METHOD PUBLIC GetSerializer : I_Serializer
VAR_INPUT
END_VAR
GetSerializer := serializer.Clone();
END_METHOD

METHOD PUBLIC RejectWithError
VAR_INPUT
	ErrorCode : T_MAXSTRING;
	Message : T_MAXSTRING;
END_VAR
serverResponse.Error(ErrorCode, Message);
END_METHOD

METHOD PUBLIC TryMakeAsynchronous : BOOL
VAR_INPUT
	Destination : REFERENCE TO I_AsynchronousRpcResponse;
END_VAR
VAR
	asynchronousRpcResponseFactory : AsynchronousRpcResponseFactory(serverResponse, serializer, asyncResponseManager);
END_VAR
TryMakeAsynchronous := asynchronousRpcResponseFactory.TryCreate(Destination);
END_METHOD

END_FUNCTION_BLOCK

// _Internal/RPC/Response/Factory/AsynchronousRpcResponseFactory
{attribute 'linkalways'} 
{attribute 'no_explicit_call' := 'This FB is a CLASS and must be accessed using methods or properties'}
{attribute 'enable_dynamic_creation'}
FUNCTION_BLOCK AsynchronousRpcResponseFactory IMPLEMENTS I_AsynchronousRpcResponseFactory
VAR
	serverResponse : I_ServerResponse;
	serializer : I_Serializer;
	asyncResponseManager : I_AsyncResponseManager;
END_VAR

METHOD FB_init : BOOL
VAR_INPUT
	bInitRetains : BOOL; // if TRUE, the retain variables are initialized (warm start / cold start)
	bInCopyCode : BOOL;  // if TRUE, the instance afterwards gets moved into the copy code (online change)
	ServerResponse : I_ServerResponse;
	Serializer : I_Serializer;
	AsyncResponseManager : I_AsyncResponseManager;
END_VAR
THIS^.serverResponse := ServerResponse;
THIS^.serializer := Serializer;
THIS^.asyncResponseManager := AsyncResponseManager;
END_METHOD

METHOD PUBLIC TryCreate : BOOL
VAR_INPUT
	Destination : REFERENCE TO I_AsynchronousRpcResponse;
END_VAR
VAR
	asyncResponseSessionData : I_AsyncResponseSessionData;
	pAsynchronousRpcResponse : POINTER TO AsynchronousRpcResponse;
END_VAR
IF NOT asyncResponseManager.TryConvertResponseToAsyncResponseSessionData(serverResponse, 0, asyncResponseSessionData) THEN
	RETURN;
END_IF

pAsynchronousRpcResponse := __NEW(AsynchronousRpcResponse(AsyncResponse := asyncResponseSessionData, Serializer := THIS^.serializer));
Destination := pAsynchronousRpcResponse^;
TryCreate := TRUE;
END_METHOD

END_FUNCTION_BLOCK

// _Internal/RPC/Response/Factory/I_AsynchronousRpcResponseFactory
INTERFACE I_AsynchronousRpcResponseFactory

METHOD PUBLIC TryCreate : BOOL
VAR_INPUT
	Destination : REFERENCE TO I_AsynchronousRpcResponse;
END_VAR
END_METHOD

END_INTERFACE

// _Internal/RPC/Middleware/RpcMiddleware
{attribute 'linkalways'} 
{attribute 'no_explicit_call' := 'This FB is a CLASS and must be accessed using methods or properties'}
{attribute 'enable_dynamic_creation'}
FUNCTION_BLOCK RpcMiddleware EXTENDS MiddlewareBase
VAR
	rpcManager : I_RpcManager;
END_VAR

METHOD FB_init : BOOL
VAR_INPUT
	bInitRetains : BOOL; // if TRUE, the retain variables are initialized (warm start / cold start)
	bInCopyCode : BOOL;  // if TRUE, the instance afterwards gets moved into the copy code (online change)
	RpcManager : I_RpcManager;
END_VAR
THIS^.rpcManager := RpcManager;
END_METHOD

METHOD PUBLIC Handle
VAR_INPUT
	Request : I_Request;
	Response : I_ServerResponse;
END_VAR
IF rpcManager.TryHandleIncomingRequest(Request, Response) THEN
	RETURN;
END_IF

Next(Request, Response);
END_METHOD

END_FUNCTION_BLOCK

// _Internal/RPC/RegisteredRpcApis/RegisteredRpcApis
{attribute 'linkalways'} 
{attribute 'no_explicit_call' := 'This FB is a CLASS and must be accessed using methods or properties'}
{attribute 'enable_dynamic_creation'}
FUNCTION_BLOCK RegisteredRpcApis
VAR
	registeredRpcApis : Queue;
	_hasRegisteredRpcApis : BOOL;
	enumerator : I_ForwardEnumerator;
END_VAR

METHOD FB_exit : BOOL
VAR_INPUT
	bInCopyCode : BOOL; // if TRUE, the exit method is called for exiting an instance that is copied afterwards (online change).
END_VAR
IF bInCopyCode THEN
	RETURN;
END_IF

IF enumerator <> 0 THEN
	enumerator.Dispose();
END_IF
END_METHOD

METHOD PRIVATE CreateEnumerator
VAR_INPUT
END_VAR
IF enumerator <> 0 THEN
	enumerator.Dispose();
END_IF

enumerator := registeredRpcApis.GetEnumerator();
END_METHOD

METHOD PUBLIC CyclicCall
VAR
	rpcApi : I_RpcApi;
END_VAR
IF NOT HasRegisteredRpcApis THEN
	RETURN;
END_IF

enumerator.Reset();

WHILE enumerator.MoveNext() DO
	IF enumerator.TryGet(rpcApi) THEN
		rpcApi.CyclicCall();
	END_IF;
END_WHILE
END_METHOD

PROPERTY PUBLIC HasRegisteredRpcApis : BOOL
GET
HasRegisteredRpcApis := enumerator <> 0;
END_GET
END_PROPERTY

METHOD PUBLIC RegisterRpcApi
VAR_INPUT
	RpcApi : I_RpcApi;
END_VAR
registeredRpcApis.Enqueue(RpcApi);
CreateEnumerator();
END_METHOD

END_FUNCTION_BLOCK

// RpcApi/I_RpcApi
INTERFACE I_RpcApi

METHOD CyclicCall
VAR_INPUT
END_VAR
END_METHOD

METHOD RegisterAsynchronousRpcHandlersWith
VAR_INPUT
	Host : I_HostAsynchronousRpcHandlers;
END_VAR
END_METHOD

METHOD RegisterSynchronousRpcHandlersWith
VAR_INPUT
	Host : I_HostSynchronousRpcHandlers;
END_VAR
END_METHOD

END_INTERFACE

// _Internal/Sessions/Manager/I_SessionManager
INTERFACE I_SessionManager

METHOD PUBLIC CreateSession : T_MAXSTRING
END_METHOD

METHOD PUBLIC DisposeAllSessions
VAR_INPUT
END_VAR
END_METHOD

METHOD PUBLIC IsValidSession : BOOL
VAR_INPUT
	Id : T_MAXSTRING;
END_VAR
END_METHOD

METHOD PUBLIC RefreshSession
VAR_INPUT
	Id : T_MAXSTRING;
END_VAR
END_METHOD

END_INTERFACE

// _Internal/Sessions/Manager/SessionManager
{attribute 'linkalways'} 
{attribute 'no_explicit_call' := 'This FB is a CLASS and must be accessed using methods or properties'}
{attribute 'enable_dynamic_creation'}
FUNCTION_BLOCK SessionManager implements I_SessionManager, I_SessionStorage
VAR
	activeSessions : Dictionary;
	sessionIdGenerator : I_SessionIdGenerator;
	currentStorageId : UDINT;
	sessionMaxLife : TIME;
END_VAR

METHOD FB_init : BOOL
VAR_INPUT
	bInitRetains : BOOL; // if TRUE, the retain variables are initialized (warm start / cold start)
	bInCopyCode : BOOL;  // if TRUE, the instance afterwards gets moved into the copy code (online change)
	SessionIdGenerator : I_SessionIdGenerator;
	SessionMaxLife : TIME;
END_VAR
THIS^.sessionIdGenerator := SessionIdGenerator;
THIS^.sessionMaxLife := SessionMaxLife;
END_METHOD

METHOD FB_exit : BOOL
VAR_INPUT
	bInCopyCode : BOOL; // if TRUE, the exit method is called for exiting an instance that is copied afterwards (online change).
END_VAR
IF bInCopyCode THEN
	RETURN;
END_IF

DisposeAllSessions();
END_METHOD

METHOD PUBLIC CheckForExpiredSessions
VAR_INPUT
END_VAR
VAR
	enumerator : I_ForwardEnumerator;
	session : I_Session;
	expiredSessions : Stack;
END_VAR
enumerator := activeSessions.GetEnumerator();

WHILE enumerator.MoveNext() DO
	IF enumerator.TryGet(session) THEN
		IF session.LastAccessedTimestamp.IsDurationElapsed(sessionMaxLife) THEN
			expiredSessions.Push(session);
		END_IF
	END_IF
END_WHILE

enumerator.Dispose();

WHILE expiredSessions.TryPop(session) DO
	DisposeSession(session.Id);
END_WHILE
END_METHOD

METHOD PRIVATE CreateNewSession : I_Session
VAR
	id : T_MAXSTRING;
	pSession : POINTER TO Session;
END_VAR
id := sessionIdGenerator.Generate();
pSession := __NEW(Session(SessionId := id));
CreateNewSession := pSession^;
END_METHOD

METHOD PUBLIC CreateSession : T_MAXSTRING;
VAR
	session : I_Session;
END_VAR
session := CreateNewSession();
activeSessions.AddOrUpdate(session.Id, session);
CreateSession := session.Id;
END_METHOD

METHOD PUBLIC CyclicCall
VAR_INPUT
END_VAR
CheckForExpiredSessions();
END_METHOD

METHOD PUBLIC DisposeAllSessions
VAR_INPUT
END_VAR
VAR
	enumerator : I_ForwardEnumerator;
	session : I_Session;
END_VAR
enumerator := activeSessions.GetEnumerator();

WHILE enumerator.MoveNext() DO
	if enumerator.TryGet(session) then
		session.Dispose();
	END_IF
END_WHILE

enumerator.Dispose();
activeSessions.Clear();
END_METHOD

METHOD PUBLIC DisposeSession
VAR_INPUT
	Id : T_MAXSTRING;
END_VAR
VAR
	session : I_Session;
END_VAR
IF NOT activeSessions.TryGetValue(Id, session) THEN
	RETURN;
END_IF

session.Dispose();
activeSessions.Remove(Id);
END_METHOD

METHOD PUBLIC DisposeSessionDataById
VAR_INPUT
	SessionId : T_MAXSTRING;
	StorageId : T_MAXSTRING;
END_VAR
VAR
	session : I_Session;
	sessionData : I_SessionData;
END_VAR
IF StorageId = '' THEN 
	RETURN;
END_IF

IF NOT activeSessions.TryGetValue(SessionId, session) THEN
	RETURN;
END_IF

IF NOT session.TryGetDataFromStorage(StorageId, sessionData) THEN
	RETURN;
END_IF

session.DisposeDataFromStorage(StorageId);
END_METHOD

METHOD PUBLIC IsValidSession : BOOL
VAR_INPUT
	Id : T_MAXSTRING;
END_VAR
IsValidSession := activeSessions.ContainsKey(Id);
END_METHOD

METHOD PUBLIC RefreshSession
VAR_INPUT
	Id : T_MAXSTRING;
END_VAR
VAR
	session : I_Session;
END_VAR
IF NOT activeSessions.TryGetValue(Id, session) THEN
	RETURN;
END_IF

session.Refresh();
END_METHOD

PROPERTY PUBLIC SessionCount : DINT
GET
SessionCount := activeSessions.Count;
END_GET
END_PROPERTY

METHOD PUBLIC TryRetreiveSessionDataById : BOOL
VAR_INPUT
	SessionId : T_MAXSTRING;
	StorageId : T_MAXSTRING;
	Destination : REFERENCE TO I_SessionData;
END_VAR
VAR
	session : I_Session;
END_VAR
IF NOT activeSessions.TryGetValue(SessionId, session) THEN
	RETURN;
END_IF

TryRetreiveSessionDataById := session.TryGetDataFromStorage(StorageId, Destination);
END_METHOD

METHOD PUBLIC TryStoreSessionDataById : BOOL
VAR_INPUT
	SessionId : T_MAXSTRING;
	StorageId : T_MAXSTRING;
	Source : I_SessionData;
END_VAR
VAR
	session : I_Session;
END_VAR
IF StorageId = '' THEN 
	RETURN;
END_IF

IF NOT activeSessions.TryGetValue(SessionId, session) THEN
	RETURN;
END_IF

session.AddOrUpdateStorage(StorageId, Source);
TryStoreSessionDataById := TRUE;
END_METHOD

END_FUNCTION_BLOCK

// _Internal/Sessions/SessionId/I_SessionIdGenerator
INTERFACE I_SessionIdGenerator

METHOD PUBLIC Generate : T_MAXSTRING
VAR_INPUT
END_VAR
END_METHOD

END_INTERFACE

// _Internal/Sessions/Middleware/SessionsMiddleware
{attribute 'linkalways'} 
{attribute 'no_explicit_call' := 'This FB is a CLASS and must be accessed using methods or properties'}
{attribute 'enable_dynamic_creation'}
FUNCTION_BLOCK SessionsMiddleware EXTENDS MiddlewareBase
VAR
	sessionManager: I_SessionManager;
	headerAccessor : I_SessionHeaderAccessor;
END_VAR

METHOD FB_init : BOOL
VAR_INPUT
	bInitRetains : BOOL; // if TRUE, the retain variables are initialized (warm start / cold start)
	bInCopyCode : BOOL;  // if TRUE, the instance afterwards gets moved into the copy code (online change)
	SessionManager : I_SessionManager;
	HeaderAccessor : I_SessionHeaderAccessor;
END_VAR
THIS^.sessionManager := SessionManager;
THIS^.headerAccessor := HeaderAccessor;
END_METHOD

METHOD PUBLIC Handle
VAR_INPUT
	Request : I_Request;
	Response : I_ServerResponse;
END_VAR
VAR
	sessionId : T_MAXSTRING;
END_VAR
IF (NOT headerAccessor.TryGetSessionIdFromRequest(Request, sessionId)) OR_ELSE (NOT sessionManager.IsValidSession(sessionId)) THEN
	sessionId := sessionManager.CreateSession();
	headerAccessor.UpdateRequestWithSessionId(Request,sessionId);
END_IF

sessionManager.RefreshSession(sessionId);

headerAccessor.UpdateResponseWithSessionId(Response, sessionId);
Next(Request, Response);
END_METHOD

END_FUNCTION_BLOCK

// _Internal/Sessions/SessionId/SequentialSessionIdGenerator
{attribute 'linkalways'} 
{attribute 'no_explicit_call' := 'This FB is a CLASS and must be accessed using methods or properties'}
{attribute 'enable_dynamic_creation'}
FUNCTION_BLOCK SequentialSessionIdGenerator Implements I_SessionIdGenerator
VAR
	currentCount : UDINT;
END_VAR

METHOD PUBLIC Generate : T_MAXSTRING
VAR_INPUT
END_VAR
currentCount := currentCount + 1;
Generate := UDINT_TO_STRING(currentCount);
END_METHOD

END_FUNCTION_BLOCK

// RpcHandler/Examples/AsyncConcatStringRpcHandler
{attribute 'linkalways'} 
FUNCTION_BLOCK AsyncConcatStringRpcHandler IMPLEMENTS I_AsynchronousRpcHandler
VAR
END_VAR

METHOD Handle
VAR_INPUT
	Parameters : I_Deserializer;
	Response : I_AsynchronousRpcResponse;
END_VAR
VAR
	str1 : T_MAXSTRING;
	str2 : T_MAXSTRING;
	result : T_MAXSTRING;
	feedback : DeserializerFeedback;
END_VAR
IF NOT Parameters.TryGetKeyString('STR1',str1,feedback) THEN
	Response.RejectWithError('MISSING_PARAMETER',feedback.FirstError.Message);
	RETURN;
END_IF

IF NOT Parameters.TryGetKeyString('STR2',str2,feedback) THEN
	Response.RejectWithError('MISSING_PARAMETER',feedback.FirstError.Message);
	RETURN;
END_IF

result := CONCAT(str1, str2);
Response.CompleteWithString(result);
END_METHOD

END_FUNCTION_BLOCK

// RpcHandler/Examples/ConcatStringRpcHandler
{attribute 'linkalways'} 
FUNCTION_BLOCK ConcatStringRpcHandler IMPLEMENTS I_SynchronousRpcHandler
VAR
END_VAR

METHOD Handle
VAR_INPUT
	Parameters : I_Deserializer;
	Response : I_SynchronousRpcResponse;
END_VAR
VAR
	str1 : T_MAXSTRING;
	str2 : T_MAXSTRING;
	result : T_MAXSTRING;
	feedback : DeserializerFeedback;
END_VAR
IF NOT Parameters.TryGetKeyString('STR1',str1,feedback) THEN
	Response.RejectWithError('MISSING_PARAMETER',feedback.FirstError.Message);
	RETURN;
END_IF

IF NOT Parameters.TryGetKeyString('STR2',str2,feedback) THEN
	Response.RejectWithError('MISSING_PARAMETER',feedback.FirstError.Message);
	RETURN;
END_IF

result := CONCAT(str1, str2);
Response.CompleteWithString(result);
END_METHOD

END_FUNCTION_BLOCK

// RpcServer/I_RpcServer
INTERFACE I_RpcServer

METHOD PUBLIC GetConfiguredHeaderSize : UDINT
VAR_INPUT
END_VAR
END_METHOD

METHOD PUBLIC GetConfiguredPayloadSize : UDINT
VAR_INPUT
END_VAR
END_METHOD

{attribute 'TcRpcEnable'}
METHOD PUBLIC HandleRequest : ResponseData;
VAR_INPUT
	SerializedHeader : STRING(ServerConfiguration.HEADER_STRING_SIZE);
	SerializedPayload : STRING(ServerConfiguration.PAYLOAD_STRING_SIZE);
END_VAR
END_METHOD

METHOD PUBLIC RegisterApi
VAR_INPUT
	RpcApi : I_RpcApi;
END_VAR
END_METHOD

METHOD PUBLIC RegisterAsynchronousRpcHandler
VAR_INPUT
	MethodName : T_MAXSTRING;
	Handler : I_AsynchronousRpcHandler;
END_VAR
END_METHOD

METHOD PUBLIC RegisterSynchronousRpcHandler
VAR_INPUT
	MethodName : T_MAXSTRING;
	Handler : I_SynchronousRpcHandler;
END_VAR
END_METHOD

END_INTERFACE

// RpcServer/RpcServer
{attribute 'linkalways'} 
{attribute 'no_explicit_call' := 'This FB is a CLASS and must be accessed using methods or properties'}
{attribute 'enable_dynamic_creation'}
{attribute 'TcRpcEnable'}
FUNCTION_BLOCK RpcServer IMPLEMENTS I_RpcServer
VAR
	// default header accessor.
	headerAccessor : HeaderAccessor;
	
	// Payload size may be changed using the constants
	payloadStringSizeIncludingNull : UDINT := ServerConfiguration.PAYLOAD_STRING_SIZE + 1;
	
	// the middleware stack allows us to construct our server in any way needed.
	// by default we will support sessions, async polling and chunked requests/
	middlewareStack : MiddlewareStack;
	
	// responseId generation required for pending or chunked data
	sequentialResponseIdGenerator : SequentialResponseIdGenerator;
	
	// ability to support sessions...
	sessionIdGenerator : SequentialSessionIdGenerator;
	sessionManager : SessionManager(sessionIdGenerator, INACTIVE_SESSION_MAX_AGE);
	sessionsMiddleware : SessionsMiddleware(sessionManager, headerAccessor);
	
	// ability to suppoort chunked requests
	chunkedRequestsManager : ChunkedRequestsManager(payloadStringSizeIncludingNull, sessionManager, headerAccessor);
	chunkedRequestsMiddleware : ChunkedRequestsMiddleware(chunkedRequestsManager);
	
	// ability to support chunked responses
	chunkedResponseManager : ChunkedResponseManager(payloadStringSizeIncludingNull, sessionManager, sequentialResponseIdGenerator, headerAccessor);
	chunkedResponsesMiddleware : ChunkedResponsesMiddleware(chunkedResponseManager);
	
	// ability to support pending responses
	asyncResponseManager : AsyncResponseManager(sessionManager, sequentialResponseIdGenerator, headerAccessor);
	asyncResponseMiddleware : AsyncResponseMiddleware(asyncResponseManager);
	
	// ability to support rpc
	synchronousRpcHandlers : SynchronousRpcHandlers;
	asynchronousRpcHandlers : AsynchronousRpcHandlers;
	asyncRpcCallQueue : AsyncRpcCallQueue;
	rpcManager : RpcManager(synchronousRpcHandlers, asynchronousRpcHandlers, asyncResponseManager, headerAccessor, asyncRpcCallQueue);
	rpcMiddleware : RpcMiddleware(rpcManager);
	
	// registered apis (used for cyclic calling)
	registeredRpcApis : RegisteredRpcApis;
	
END_VAR
VAR CONSTANT
	INACTIVE_SESSION_MAX_AGE : TIME := T#10S;
END_VAR

METHOD FB_init : BOOL
VAR_INPUT
	bInitRetains : BOOL; // if TRUE, the retain variables are initialized (warm start / cold start)
	bInCopyCode : BOOL;  // if TRUE, the instance afterwards gets moved into the copy code (online change)
END_VAR
// must be above any middleware which requires storing of session data. 
// best practice is to put at the top
MiddlewareStack.Use(sessionsMiddleware);

// must be above any middleware which could send a response larger than the max payload.
// once this is in place then middleware can send as large as they like (up to router memory max)
MiddlewareStack.Use(chunkedResponsesMiddleware);

// must be above any middleware which needs to support async responses
MiddlewareStack.Use(AsyncResponseMiddleware);

// chunked request must be after chunked response to prevent incorrectly starting a new request
// if the client askes for a response without removing the last request header.
MiddlewareStack.Use(chunkedRequestsMiddleware); 

// rpc middlware.  All other middleware can go under here.
MiddlewareStack.Use(rpcMiddleware);
END_METHOD

METHOD PUBLIC CyclicCall
VAR_INPUT
END_VAR
sessionManager.CyclicCall();
asyncRpcCallQueue.CyclicCall();
registeredRpcApis.CyclicCall();
END_METHOD

{attribute 'TcRpcEnable'}
METHOD PUBLIC GetConfiguredHeaderSize : UDINT
VAR_INPUT
END_VAR
GetConfiguredHeaderSize := ServerConfiguration.HEADER_STRING_SIZE;
END_METHOD

{attribute 'TcRpcEnable'}
METHOD PUBLIC GetConfiguredPayloadSize : UDINT
VAR_INPUT
END_VAR
GetConfiguredPayloadSize := ServerConfiguration.PAYLOAD_STRING_SIZE;
END_METHOD

{attribute 'TcRpcEnable'}
METHOD PUBLIC HandleRequest : ResponseData;
VAR_INPUT
	SerializedHeader : STRING(ServerConfiguration.HEADER_STRING_SIZE);
	SerializedPayload : STRING(ServerConfiguration.PAYLOAD_STRING_SIZE);
END_VAR
VAR
	header : Header(SerializedHeader);
	request : Request(header, SerializedPayload);
	serverResponse : ServerResponse(headerAccessor);
END_VAR
middlewareStack.Handle(request, serverResponse);

IF NOT serverResponse.HeadersSent THEN
	serverResponse.Error('UNHANDLED_REQUEST', 'Unhandled Request');
END_IF

serverResponse.TryGetData(HandleRequest);
END_METHOD

METHOD PUBLIC RegisterApi
VAR_INPUT
	RpcApi : I_RpcApi;
END_VAR
RpcApi.RegisterSynchronousRpcHandlersWith(synchronousRpcHandlers);
RpcApi.RegisterAsynchronousRpcHandlersWith(asynchronousRpcHandlers);
registeredRpcApis.RegisterRpcApi(RpcApi);
END_METHOD

METHOD PUBLIC RegisterAsynchronousRpcHandler
VAR_INPUT
	MethodName : T_MAXSTRING;
	Handler : I_AsynchronousRpcHandler;
END_VAR
asynchronousRpcHandlers.RegisterHandler(MethodName, Handler);
END_METHOD

METHOD PUBLIC RegisterSynchronousRpcHandler
VAR_INPUT
	MethodName : T_MAXSTRING;
	Handler : I_SynchronousRpcHandler;
END_VAR
synchronousRpcHandlers.RegisterHandler(MethodName, Handler);
END_METHOD

PROPERTY PUBLIC SessionCount : DINT
GET
SessionCount := sessionManager.SessionCount;
END_GET
END_PROPERTY

METHOD PUBLIC Use
VAR_INPUT
	Middleware : I_Middleware;
END_VAR
middlewareStack.Use(Middleware);
END_METHOD

END_FUNCTION_BLOCK
